// TIA Portal V17 export
// export: Created 2023-02-26T22:27:32.0311882Z, ExportSetting WithDefaults, DisplayName Totally Integrated Automation Portal, DisplayVersion V17, DisplayName TIA Portal Openness, DisplayVersion V17, DisplayName TIA Portal Version Control Interface, DisplayVersion V17, DisplayName TIA Portal Test Suite Advanced, DisplayVersion V17, DisplayName STEP 7 Professional, DisplayVersion V17, DisplayName SIMATIC Energy Suite, DisplayVersion V17, DisplayName STEP 7 Safety, DisplayVersion V17, DisplayName WinCC Professional, DisplayVersion V17
TYPE "stt_LostPackageError"
// stored: IsFailsafeCompliant false
   STRUCT
      Error_1 : Bool;
      Error_2 : Bool;
      Error_3 : Bool;
      Error_4 : Bool;
      Error_5 : Bool;
      Error_6 : Bool;
   END_STRUCT;
END_TYPE
